    conveyors/product_killer2/status_act_prod AT 723 : DINT := 0;
    conveyors/product_killer2/m11 AT 7168 : REAL := 30.9461;
    conveyors/product_killer2/m12 AT 7169 : REAL := 0.0;
    conveyors/product_killer2/m13 AT 7170 : REAL := 0.0;
    conveyors/product_killer2/m14 AT 7171 : REAL := 935.942;
    conveyors/product_killer2/m21 AT 7172 : REAL := 0.0;
    conveyors/product_killer2/m22 AT 7173 : REAL := 33.1565;
    conveyors/product_killer2/m23 AT 7174 : REAL := 0.0;
    conveyors/product_killer2/m24 AT 7175 : REAL := 410.0;
    conveyors/product_killer2/m31 AT 7176 : REAL := 0.0;
    conveyors/product_killer2/m32 AT 7177 : REAL := 0.0;
    conveyors/product_killer2/m33 AT 7178 : REAL := 12.0;
    conveyors/product_killer2/m34 AT 7179 : REAL := 428.0;
    conveyors/product_killer2/m41 AT 7180 : REAL := 0.0;
    conveyors/product_killer2/m42 AT 7181 : REAL := 0.0;
    conveyors/product_killer2/m43 AT 7182 : REAL := 0.0;
    conveyors/product_killer2/m44 AT 7183 : REAL := 1.0;
    conveyors/product_killer2/isActive AT 405 : BOOL := true;
    conveyors/ejector/energy AT 349 : BOOL := true;
    conveyors/ejector/cmdSupply AT 348 : BOOL := true;
    conveyors/ejector/sensorSupply AT 347 : BOOL := true;
    conveyors/ejector/valveWork AT 29 : BOOL := false;
    conveyors/ejector/outletSensor AT 346 : BOOL := false;
    conveyors/ejector/inletSensor AT 345 : BOOL := false;
    conveyors/ejector/rodPosition AT 7117 : REAL := 0.0;
    conveyors/ejector/rodPercent AT 7116 : REAL := 0.0;
    conveyors/ejector/incrementValue AT 7122 : REAL := 0.0;
    conveyors/ejector/slidePosition AT 724 : DINT := 0;
    conveyors/ejector/pipeWork AT 406 : BOOL := false;
    conveyors/ejector/pipeRest AT 407 : BOOL := false;
    conveyors/ejector/increment AT 7184 : REAL := 0.0;
    conveyors/ejector/outletSensorLogic AT 408 : BOOL := true;
    conveyors/ejector/inletSensorLogic AT 409 : BOOL := true;
    conveyors/ejector/rodLength AT 7185 : REAL := 360.0;
    conveyors/ejector/time2extend AT 7186 : REAL := 2.0;
    conveyors/ejector/d_locking AT 410 : BOOL := false;
    conveyors/ejector/v_d_locking AT 7187 : REAL := 2.0;
    conveyors/ejector/d_inletSensor AT 411 : BOOL := false;
    conveyors/ejector/v_d_inletSensor AT 412 : BOOL := false;
    conveyors/ejector/d_outletSensor AT 413 : BOOL := false;
    conveyors/ejector/v_d_outletSensor AT 414 : BOOL := false;
    conveyors/qrreader1/idRead AT 525 : INT := 0;
    conveyors/qrreader1/status_act_prod AT 725 : DINT := 0;
    conveyors/qrreader1/m11 AT 7188 : REAL := 73.8285;
    conveyors/qrreader1/m12 AT 7189 : REAL := 0.0;
    conveyors/qrreader1/m13 AT 7190 : REAL := 0.0;
    conveyors/qrreader1/m14 AT 7191 : REAL := 938.152;
    conveyors/qrreader1/m21 AT 7192 : REAL := 0.0;
    conveyors/qrreader1/m22 AT 7193 : REAL := 80.0;
    conveyors/qrreader1/m23 AT 7194 : REAL := 0.0;
    conveyors/qrreader1/m24 AT 7195 : REAL := 810.0;
    conveyors/qrreader1/m31 AT 7196 : REAL := 0.0;
    conveyors/qrreader1/m32 AT 7197 : REAL := 0.0;
    conveyors/qrreader1/m33 AT 7198 : REAL := 70.0;
    conveyors/qrreader1/m34 AT 7199 : REAL := 420.0;
    conveyors/qrreader1/m41 AT 7200 : REAL := 0.0;
    conveyors/qrreader1/m42 AT 7201 : REAL := 0.0;
    conveyors/qrreader1/m43 AT 7202 : REAL := 0.0;
    conveyors/qrreader1/m44 AT 7203 : REAL := 1.0;
    conveyors/qrreader1/number AT 726 : INT := 0;
    conveyors/weighingscale1/Weight AT 526 : INT := 0;
    conveyors/weighingscale1/status_act_prod AT 727 : DINT := 0;
    conveyors/weighingscale1/m11 AT 7204 : REAL := 87.9752;
    conveyors/weighingscale1/m12 AT 7205 : REAL := 0.0;
    conveyors/weighingscale1/m13 AT 7206 : REAL := 0.0;
    conveyors/weighingscale1/m14 AT 7207 : REAL := 870.0;
    conveyors/weighingscale1/m21 AT 7208 : REAL := 0.0;
    conveyors/weighingscale1/m22 AT 7209 : REAL := 44.2087;
    conveyors/weighingscale1/m23 AT 7210 : REAL := 0.0;
    conveyors/weighingscale1/m24 AT 7211 : REAL := 575.0;
    conveyors/weighingscale1/m31 AT 7212 : REAL := 0.0;
    conveyors/weighingscale1/m32 AT 7213 : REAL := 0.0;
    conveyors/weighingscale1/m33 AT 7214 : REAL := 70.0;
    conveyors/weighingscale1/m34 AT 7215 : REAL := 420.0;
    conveyors/weighingscale1/m41 AT 7216 : REAL := 0.0;
    conveyors/weighingscale1/m42 AT 7217 : REAL := 0.0;
    conveyors/weighingscale1/m43 AT 7218 : REAL := 0.0;
    conveyors/weighingscale1/m44 AT 7219 : REAL := 1.0;
    conveyors/weighingscale1/weight AT 728 : INT := 0;
    conveyors/prdEndConvUp/incPositionX AT 7115 : REAL := 0.0;
    conveyors/prdEndConvUp/incPositionY AT 7114 : REAL := 0.0;
    conveyors/prdEndConvUp/incPositionZ AT 7113 : REAL := 0.0;
    conveyors/prdEndConvUp/coordCenterX AT 7112 : REAL := 0.0;
    conveyors/prdEndConvUp/coordCenterY AT 7111 : REAL := 0.0;
    conveyors/prdEndConvUp/coordCenterZ AT 7110 : REAL := 0.0;
    conveyors/prdEndConvUp/incRotationX AT 7109 : REAL := 0.0;
    conveyors/prdEndConvUp/incRotationY AT 7108 : REAL := 0.0;
    conveyors/prdEndConvUp/incRotationZ AT 7107 : REAL := 0.0;
    conveyors/prdEndConvUp/sensorSupply AT 344 : BOOL := true;
    conveyors/prdEndConvUp/presence AT 6 : BOOL := false;
    conveyors/prdEndConvUp/status_act_prod AT 729 : DINT := 0;
    conveyors/prdEndConvUp/m11 AT 7220 : REAL := 0.0;
    conveyors/prdEndConvUp/m12 AT 7221 : REAL := -199.823;
    conveyors/prdEndConvUp/m13 AT 7222 : REAL := 0.0;
    conveyors/prdEndConvUp/m14 AT 7223 : REAL := 814.81;
    conveyors/prdEndConvUp/m21 AT 7224 : REAL := 12.8205;
    conveyors/prdEndConvUp/m22 AT 7225 : REAL := 0.0;
    conveyors/prdEndConvUp/m23 AT 7226 : REAL := 0.0;
    conveyors/prdEndConvUp/m24 AT 7227 : REAL := 893.28;
    conveyors/prdEndConvUp/m31 AT 7228 : REAL := 0.0;
    conveyors/prdEndConvUp/m32 AT 7229 : REAL := 0.0;
    conveyors/prdEndConvUp/m33 AT 7230 : REAL := 14.1468;
    conveyors/prdEndConvUp/m34 AT 7231 : REAL := 680.0;
    conveyors/prdEndConvUp/m41 AT 7232 : REAL := 0.0;
    conveyors/prdEndConvUp/m42 AT 7233 : REAL := 0.0;
    conveyors/prdEndConvUp/m43 AT 7234 : REAL := 0.0;
    conveyors/prdEndConvUp/m44 AT 7235 : REAL := 1.0;
    conveyors/prdEndConvUp/detection AT 415 : BOOL := false;
    conveyors/prdEndConvUp/presenceLogic AT 416 : BOOL := true;
    conveyors/prdEndConvUp/d_presence AT 417 : BOOL := false;
    conveyors/prdEndConvUp/v_d_presence AT 418 : BOOL := true;
    conveyors/prdBegConvDw/incPositionX AT 7106 : REAL := 0.0;
    conveyors/prdBegConvDw/incPositionY AT 7105 : REAL := 0.0;
    conveyors/prdBegConvDw/incPositionZ AT 7104 : REAL := 0.0;
    conveyors/prdBegConvDw/coordCenterX AT 7103 : REAL := 0.0;
    conveyors/prdBegConvDw/coordCenterY AT 7102 : REAL := 0.0;
    conveyors/prdBegConvDw/coordCenterZ AT 7101 : REAL := 0.0;
    conveyors/prdBegConvDw/incRotationX AT 7100 : REAL := 0.0;
    conveyors/prdBegConvDw/incRotationY AT 7099 : REAL := 0.0;
    conveyors/prdBegConvDw/incRotationZ AT 7098 : REAL := 0.0;
    conveyors/prdBegConvDw/sensorSupply AT 343 : BOOL := true;
    conveyors/prdBegConvDw/presence AT 7 : BOOL := false;
    conveyors/prdBegConvDw/status_act_prod AT 730 : DINT := 0;
    conveyors/prdBegConvDw/m11 AT 7236 : REAL := 12.8205;
    conveyors/prdBegConvDw/m12 AT 7237 : REAL := 0.0;
    conveyors/prdBegConvDw/m13 AT 7238 : REAL := 0.0;
    conveyors/prdBegConvDw/m14 AT 7239 : REAL := 940.0;
    conveyors/prdBegConvDw/m21 AT 7240 : REAL := 0.0;
    conveyors/prdBegConvDw/m22 AT 7241 : REAL := 200.0;
    conveyors/prdBegConvDw/m23 AT 7242 : REAL := 0.0;
    conveyors/prdBegConvDw/m24 AT 7243 : REAL := 615.0;
    conveyors/prdBegConvDw/m31 AT 7244 : REAL := 0.0;
    conveyors/prdBegConvDw/m32 AT 7245 : REAL := 0.0;
    conveyors/prdBegConvDw/m33 AT 7246 : REAL := 12.8205;
    conveyors/prdBegConvDw/m34 AT 7247 : REAL := 428.028;
    conveyors/prdBegConvDw/m41 AT 7248 : REAL := 0.0;
    conveyors/prdBegConvDw/m42 AT 7249 : REAL := 0.0;
    conveyors/prdBegConvDw/m43 AT 7250 : REAL := 0.0;
    conveyors/prdBegConvDw/m44 AT 7251 : REAL := 1.0;
    conveyors/prdBegConvDw/detection AT 419 : BOOL := false;
    conveyors/prdBegConvDw/presenceLogic AT 420 : BOOL := true;
    conveyors/prdBegConvDw/d_presence AT 421 : BOOL := false;
    conveyors/prdBegConvDw/v_d_presence AT 422 : BOOL := true;
    conveyors/conveyorUp/incPositionX AT 7097 : REAL := 0.0;
    conveyors/conveyorUp/incPositionY AT 7096 : REAL := 0.0;
    conveyors/conveyorUp/incPositionZ AT 7095 : REAL := 0.0;
    conveyors/conveyorUp/coordCenterX AT 7094 : REAL := 0.0;
    conveyors/conveyorUp/coordCenterY AT 7093 : REAL := 0.0;
    conveyors/conveyorUp/coordCenterZ AT 7092 : REAL := 0.0;
    conveyors/conveyorUp/incRotationX AT 7091 : REAL := 0.0;
    conveyors/conveyorUp/incRotationY AT 7090 : REAL := 0.0;
    conveyors/conveyorUp/incRotationZ AT 7089 : REAL := 0.0;
    conveyors/conveyorUp/linearSpeed AT 7120 : REAL := 0.0;
    conveyors/conveyorUp/status_act_prod AT 731 : DINT := 0;
    conveyors/conveyorUp/m11 AT 7252 : REAL := 0.0;
    conveyors/conveyorUp/m12 AT 7253 : REAL := -200.0;
    conveyors/conveyorUp/m13 AT 7254 : REAL := 0.0;
    conveyors/conveyorUp/m14 AT 7255 : REAL := 815.0;
    conveyors/conveyorUp/m21 AT 7256 : REAL := 400.0;
    conveyors/conveyorUp/m22 AT 7257 : REAL := 0.0;
    conveyors/conveyorUp/m23 AT 7258 : REAL := 0.0;
    conveyors/conveyorUp/m24 AT 7259 : REAL := 850.0;
    conveyors/conveyorUp/m31 AT 7260 : REAL := 0.0;
    conveyors/conveyorUp/m32 AT 7261 : REAL := 0.0;
    conveyors/conveyorUp/m33 AT 7262 : REAL := 10.0;
    conveyors/conveyorUp/m34 AT 7263 : REAL := 665.0;
    conveyors/conveyorUp/m41 AT 7264 : REAL := 0.0;
    conveyors/conveyorUp/m42 AT 7265 : REAL := 0.0;
    conveyors/conveyorUp/m43 AT 7266 : REAL := 0.0;
    conveyors/conveyorUp/m44 AT 7267 : REAL := 1.0;
    conveyors/conveyorUp/incrementPositionX AT 7268 : REAL := 0.0;
    conveyors/conveyorUp/incrementPositionY AT 7269 : REAL := 0.0;
    conveyors/conveyorUp/incrementPositionZ AT 7270 : REAL := 0.0;
    conveyors/conveyorUp/incShiftProduct AT 7271 : REAL := 0.0;
    conveyors/conveyorUp/centerRotX AT 7272 : REAL := 0.0;
    conveyors/conveyorUp/centerRotY AT 7273 : REAL := 0.0;
    conveyors/conveyorUp/centerRotZ AT 7274 : REAL := 0.0;
    conveyors/conveyorUp/incRotY AT 7275 : REAL := 0.0;
    conveyors/conveyorUp/incRotZ AT 7276 : REAL := 0.0;
    conveyors/conveyorUp/incRotX AT 7277 : REAL := 0.0;
    conveyors/conveyorUp/d_locking AT 423 : BOOL := false;
    conveyors/conveyorUp/v_d_locking AT 424 : BOOL := false;
    conveyors/conveyorDown/incPositionX AT 7088 : REAL := 0.0;
    conveyors/conveyorDown/incPositionY AT 7087 : REAL := 0.0;
    conveyors/conveyorDown/incPositionZ AT 7086 : REAL := 0.0;
    conveyors/conveyorDown/coordCenterX AT 7085 : REAL := 0.0;
    conveyors/conveyorDown/coordCenterY AT 7084 : REAL := 0.0;
    conveyors/conveyorDown/coordCenterZ AT 7083 : REAL := 0.0;
    conveyors/conveyorDown/incRotationX AT 7082 : REAL := 0.0;
    conveyors/conveyorDown/incRotationY AT 7081 : REAL := 0.0;
    conveyors/conveyorDown/incRotationZ AT 7080 : REAL := 0.0;
    conveyors/conveyorDown/linearSpeed AT 7121 : REAL := 0.0;
    conveyors/conveyorDown/status_act_prod AT 732 : DINT := 0;
    conveyors/conveyorDown/m11 AT 7278 : REAL := 359.859;
    conveyors/conveyorDown/m12 AT 7279 : REAL := 0.0;
    conveyors/conveyorDown/m13 AT 7280 : REAL := 0.0;
    conveyors/conveyorDown/m14 AT 7281 : REAL := 919.805;
    conveyors/conveyorDown/m21 AT 7282 : REAL := 0.0;
    conveyors/conveyorDown/m22 AT 7283 : REAL := 199.823;
    conveyors/conveyorDown/m23 AT 7284 : REAL := 0.0;
    conveyors/conveyorDown/m24 AT 7285 : REAL := 615.0;
    conveyors/conveyorDown/m31 AT 7286 : REAL := 0.0;
    conveyors/conveyorDown/m32 AT 7287 : REAL := 0.0;
    conveyors/conveyorDown/m33 AT 7288 : REAL := 10.168;
    conveyors/conveyorDown/m34 AT 7289 : REAL := 419.629;
    conveyors/conveyorDown/m41 AT 7290 : REAL := 0.0;
    conveyors/conveyorDown/m42 AT 7291 : REAL := 0.0;
    conveyors/conveyorDown/m43 AT 7292 : REAL := 0.0;
    conveyors/conveyorDown/m44 AT 7293 : REAL := 1.0;
    conveyors/conveyorDown/incrementPositionX AT 7294 : REAL := 0.0;
    conveyors/conveyorDown/incrementPositionY AT 7295 : REAL := 0.0;
    conveyors/conveyorDown/incrementPositionZ AT 7296 : REAL := 0.0;
    conveyors/conveyorDown/incShiftProduct AT 7297 : REAL := 0.0;
    conveyors/conveyorDown/centerRotX AT 7298 : REAL := 0.0;
    conveyors/conveyorDown/centerRotY AT 7299 : REAL := 0.0;
    conveyors/conveyorDown/centerRotZ AT 7300 : REAL := 0.0;
    conveyors/conveyorDown/incRotY AT 7301 : REAL := 0.0;
    conveyors/conveyorDown/incRotZ AT 7302 : REAL := 0.0;
    conveyors/conveyorDown/incRotX AT 7303 : REAL := 0.0;
    conveyors/conveyorDown/d_locking AT 425 : BOOL := false;
    conveyors/conveyorDown/v_d_locking AT 426 : BOOL := false;
    conveyors/pusher1/moveX AT 7079 : REAL := 0.0;
    conveyors/pusher1/moveY AT 7122 : REAL := 0.0;
    conveyors/pusher1/moveZ AT 7078 : REAL := 0.0;
    conveyors/pusher1/status_act_prod AT 733 : DINT := 0;
    conveyors/pusher1/m11 AT 7304 : REAL := -23.4306;
    conveyors/pusher1/m12 AT 7305 : REAL := 0.0;
    conveyors/pusher1/m13 AT 7306 : REAL := 0.0;
    conveyors/pusher1/m14 AT 7307 : REAL := 973.961;
    conveyors/pusher1/m21 AT 7308 : REAL := 0.0;
    conveyors/pusher1/m22 AT 7309 : REAL := -22.1043;
    conveyors/pusher1/m23 AT 7310 : REAL := 0.0;
    conveyors/pusher1/m24 AT 7311 : REAL := 845.093;
    conveyors/pusher1/m31 AT 7312 : REAL := 0.0;
    conveyors/pusher1/m32 AT 7313 : REAL := 0.0;
    conveyors/pusher1/m33 AT 7314 : REAL := 12.0;
    conveyors/pusher1/m34 AT 7315 : REAL := 428.0;
    conveyors/pusher1/m41 AT 7316 : REAL := 0.0;
    conveyors/pusher1/m42 AT 7317 : REAL := 0.0;
    conveyors/pusher1/m43 AT 7318 : REAL := 0.0;
    conveyors/pusher1/m44 AT 7319 : REAL := 1.0;
    conveyors/pusher1/moveX1 AT 7320 : REAL := 0.0;
    conveyors/pusher1/moveY1 AT 7321 : REAL := 0.0;
    conveyors/pusher1/moveZ1 AT 7322 : REAL := 0.0;
    conveyors/pusher1/oriX AT 7323 : REAL := 1.0;
    conveyors/pusher1/oriY AT 7324 : REAL := -1.0;
    conveyors/pusher1/oriZ AT 7325 : REAL := 1.0;
  END_VAR
END_CONFIGURATION
